VISUALIZATION RightRobotStats  // 2x2
END_VISUALIZATION

(* stored: Version 1.1.0.1, ProductVersion 3.1.4024.15
   Visu RightRobotStats: Id {2e140c51-3b7c-48bb-9e9f-e8cdcecd5dd8} *)
